// TIA Portal V20 export
DATA_BLOCK "SP201"   // DB235
// stored: MemoryReserve 100
   VAR
      "MAIN OP AUTO INITIATE PBL (GREEN)" : Bool := FALSE;
      "MAIN OP STOP PBL (RED)" : Bool := FALSE;
      SPARE_5 : Bool := FALSE;
      SPARE : Bool := FALSE;
      SPARE_1 : Bool := FALSE;
      SPARE_2 : Bool := FALSE;
      SPARE_3 : Bool := FALSE;
      SPARE_4 : Bool := FALSE;
      "MAIN HMI POWER TRIPPED E110CB" : Bool := TRUE;
   END_VAR
BEGIN
END_DATA_BLOCK
